// Mitsubishi GX Works2 project: mitsubishi_fx3u_gxsimulator2   PLC: FX3U/FX3UC

PROGRAM MAIN
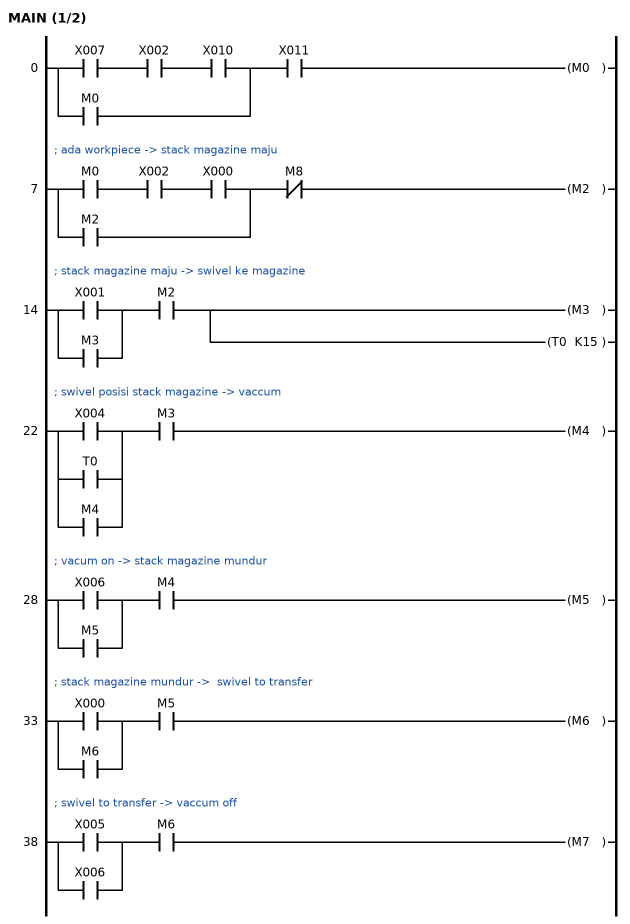
0     LD      X007
      AND     X002
      AND     X010
      OR      M0
      AND     X011
      OUT     M0
; ada workpiece -> stack magazine maju
7     LD      M0
      AND     X002
      AND     X000
      OR      M2
      ANI     M8
      OUT     M2
; stack magazine maju -> swivel ke magazine
14    LD      X001
      OR      M3
      AND     M2
      OUT     M3
      OUT     T0 K15
; swivel posisi stack magazine -> vaccum
22    LD      X004
      OR      T0
      OR      M4
      AND     M3
      OUT     M4
; vacum on -> stack magazine mundur
28    LD      X006
      OR      M5
      AND     M4
      OUT     M5
; stack magazine mundur ->  swivel to transfer
33    LD      X000
      OR      M6
      AND     M5
      OUT     M6
; swivel to transfer -> vaccum off
38    LD      X005
      OR      X006
      AND     M6
      OUT     M7
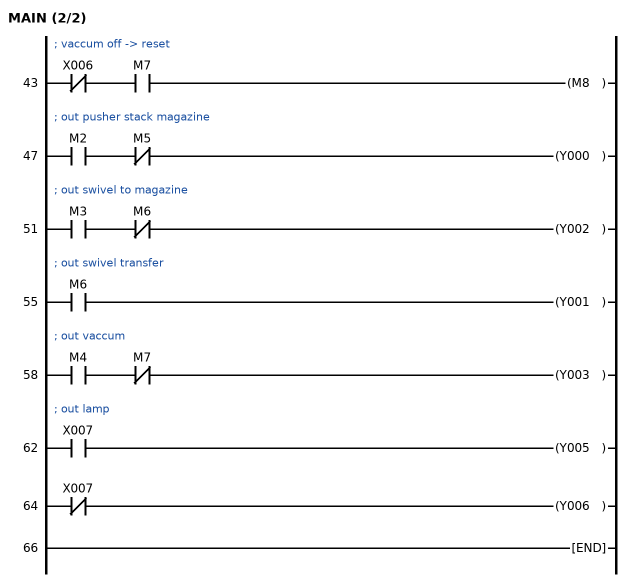
; vaccum off -> reset
43    LDI     X006
      AND     M7
      OUT     M8
; out pusher stack magazine
47    LD      M2
      ANI     M5
      OUT     Y000
; out swivel to magazine
51    LD      M3
      ANI     M6
      OUT     Y002
; out swivel transfer
55    LD      M6
      OUT     Y001
; out vaccum
58    LD      M4
      ANI     M7
      OUT     Y003
; out lamp
62    LD      X007
      OUT     Y005
64    LDI     X007
      OUT     Y006
66    END
END_PROGRAM
